FUNCTION_BLOCK SS5_ps_Ejector (* Composite FB wrapping other FBs *)
  (* Standard: 61499-2 *)
  (* Version 1.0, 2025-08-25, PS_Transformer_for_Unknown *)
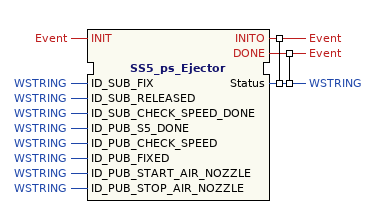
  EVENT_INPUT
    INIT; (* Initialization Request *)
  END_EVENT
  EVENT_OUTPUT
    INITO WITH Status; (* Initialization Confirm *)
    DONE WITH Status; (* Execution Confirmation *)
  END_EVENT
  VAR_INPUT
    ID_SUB_FIX : WSTRING;
    ID_SUB_RELEASED : WSTRING;
    ID_SUB_CHECK_SPEED_DONE : WSTRING;
    ID_PUB_S5_DONE : WSTRING;
    ID_PUB_CHECK_SPEED : WSTRING;
    ID_PUB_FIXED : WSTRING;
    ID_PUB_START_AIR_NOZZLE : WSTRING;
    ID_PUB_STOP_AIR_NOZZLE : WSTRING;
  END_VAR
  VAR_OUTPUT
    Status : WSTRING; (* Output event qualifier *)
  END_VAR
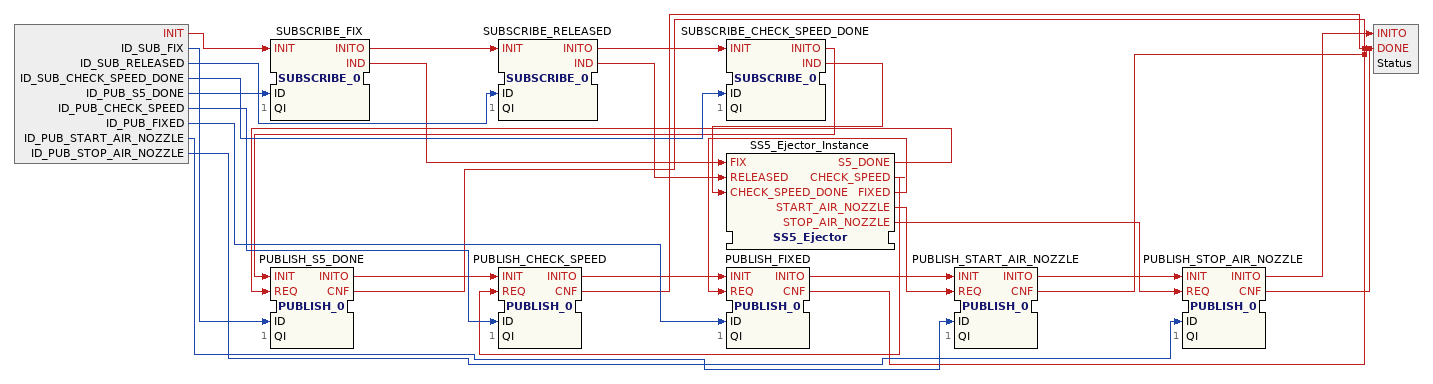
  FBS
    SS5_Ejector_Instance : SS5_Ejector;
    SUBSCRIBE_FIX : SUBSCRIBE_0(QI := 1);
    SUBSCRIBE_RELEASED : SUBSCRIBE_0(QI := 1);
    SUBSCRIBE_CHECK_SPEED_DONE : SUBSCRIBE_0(QI := 1);
    PUBLISH_S5_DONE : PUBLISH_0(QI := 1);
    PUBLISH_CHECK_SPEED : PUBLISH_0(QI := 1);
    PUBLISH_FIXED : PUBLISH_0(QI := 1);
    PUBLISH_START_AIR_NOZZLE : PUBLISH_0(QI := 1);
    PUBLISH_STOP_AIR_NOZZLE : PUBLISH_0(QI := 1);
  END_FBS
  EVENT_CONNECTIONS
    INIT TO SUBSCRIBE_FIX.INIT;
    SUBSCRIBE_FIX.INITO TO SUBSCRIBE_RELEASED.INIT;
    SUBSCRIBE_RELEASED.INITO TO SUBSCRIBE_CHECK_SPEED_DONE.INIT;
    SUBSCRIBE_CHECK_SPEED_DONE.INITO TO PUBLISH_S5_DONE.INIT;
    PUBLISH_S5_DONE.INITO TO PUBLISH_CHECK_SPEED.INIT;
    PUBLISH_CHECK_SPEED.INITO TO PUBLISH_FIXED.INIT;
    PUBLISH_FIXED.INITO TO PUBLISH_START_AIR_NOZZLE.INIT;
    PUBLISH_START_AIR_NOZZLE.INITO TO PUBLISH_STOP_AIR_NOZZLE.INIT;
    PUBLISH_STOP_AIR_NOZZLE.INITO TO INITO;
    SUBSCRIBE_FIX.IND TO SS5_Ejector_Instance.FIX;
    SUBSCRIBE_RELEASED.IND TO SS5_Ejector_Instance.RELEASED;
    SUBSCRIBE_CHECK_SPEED_DONE.IND TO SS5_Ejector_Instance.CHECK_SPEED_DONE;
    SS5_Ejector_Instance.S5_DONE TO PUBLISH_S5_DONE.REQ;
    SS5_Ejector_Instance.CHECK_SPEED TO PUBLISH_CHECK_SPEED.REQ;
    SS5_Ejector_Instance.FIXED TO PUBLISH_FIXED.REQ;
    SS5_Ejector_Instance.START_AIR_NOZZLE TO PUBLISH_START_AIR_NOZZLE.REQ;
    SS5_Ejector_Instance.STOP_AIR_NOZZLE TO PUBLISH_STOP_AIR_NOZZLE.REQ;
    PUBLISH_S5_DONE.CNF TO DONE;
    PUBLISH_CHECK_SPEED.CNF TO DONE;
    PUBLISH_FIXED.CNF TO DONE;
    PUBLISH_START_AIR_NOZZLE.CNF TO DONE;
    PUBLISH_STOP_AIR_NOZZLE.CNF TO DONE;
  END_CONNECTIONS
  DATA_CONNECTIONS
    ID_SUB_FIX TO SUBSCRIBE_FIX.ID;
    ID_SUB_RELEASED TO SUBSCRIBE_RELEASED.ID;
    ID_SUB_CHECK_SPEED_DONE TO SUBSCRIBE_CHECK_SPEED_DONE.ID;
    ID_PUB_S5_DONE TO PUBLISH_S5_DONE.ID;
    ID_PUB_CHECK_SPEED TO PUBLISH_CHECK_SPEED.ID;
    ID_PUB_FIXED TO PUBLISH_FIXED.ID;
    ID_PUB_START_AIR_NOZZLE TO PUBLISH_START_AIR_NOZZLE.ID;
    ID_PUB_STOP_AIR_NOZZLE TO PUBLISH_STOP_AIR_NOZZLE.ID;
  END_CONNECTIONS
END_FUNCTION_BLOCK
